TYPE ST_DriverAX8206_HWI :
STRUCT
  comState          : ST_CardState_HWI;
  sdiDcOutputShift  : DINT;
  sdiDcInputShift   : DINT;

  siFrontIGBTTemp   : INT;//ChB
  siBackIGBTTemp    : INT;//ChA
  
  rFrontMotorTemp  : REAL;//ChB
  rBackMotorTemp   : REAL;//ChA
  
  rFrontMotorTorque : REAL;//ChB
  rBackMotorTorque  : REAL;//ChA
  
  udFrontMotorDIGIns: UDINT;//ChB
  udBackMotorDIGIns: UDINT;//ChA
END_STRUCT
END_TYPE

(* stored: Version 1.1.0.1, ProductVersion 3.1.4024.12
   DUT ST_DriverAX8206_HWI: Id {a902e78f-3499-42e9-865a-5896e341dd21} *)
